// TIA Portal V17 export
// export: Created 2022-07-20T06:59:50.029013Z, ExportSetting WithDefaults, DisplayName Totally Integrated Automation Portal, DisplayVersion V17, DisplayName TIA Portal Openness, DisplayVersion V17, DisplayName TIA Portal Version Control Interface, DisplayVersion V17, DisplayName SINAMICS Startdrive Advanced, DisplayVersion V17, DisplayName SINAMICS Startdrive G130, G150, S120, S150, SINAMICS MV, S210, DisplayVersion V17, DisplayName SINAMICS Startdrive G110M, G120, G120C, G120D, G120P, G115D, DisplayVersion V17, DisplayName STEP 7 Professional, DisplayVersion V17, DisplayName STEP 7 Safety, DisplayVersion V17, DisplayName WinCC Advanced, DisplayVersion V17
FUNCTION "FC10028_FirstBitActivatedInValue" : SInt   // FC10028, LAD
{ S7_Optimized_Access := 'TRUE' }
VERSION : 0.1
// stored: AutoNumber false, IsIECCheckEnabled false, SetENOAutomatically false, UDAEnableTagReadback false
   VAR_INPUT
      DWord_In : DWord;
   END_VAR
   VAR_TEMP
      i : SInt;
      DWord_Temp : DWord;
   END_VAR
BEGIN

REGION Network 1 (SCL)
   IF #DWord_In <> 16#0 THEN
       #i := 0;
       #DWord_Temp := #DWord_In;
       WHILE #DWord_Temp <> 16#1 DO
           IF (#DWord_Temp MOD 16#2) = 1 THEN
               EXIT;
           ELSE
               #i += 1;
               #DWord_Temp /= 16#2;
           END_IF;
       END_WHILE;
       #FC10028_FirstBitActivatedInValue := #i;
   ELSE
       #FC10028_FirstBitActivatedInValue := -1;
   END_IF;
END_REGION
END_FUNCTION
